// SIMATIC S7-200 project (STEP 7-Micro/WIN), CPU 222 REL 02.01

SYMBOL_TABLE USER1
CASSA_PIENA      C1       // CONTEGGIO DELLE DODICI BOTTIGLIE
FC_SUP           I0.0     // FINECORSA SUPERIORE
FC_INF           I0.1     // FINECORSA INFERIORE
FC_POS           I0.2     // SENSORE DI POSIZIONE
START            I0.3     // PULSANTE AVVIO CICLO
CONT             I0.4     // DISPOSITIVO CONTEGGIO BOTTIGLIE
IN_RIEMP         M0.0     // FASE DI RIEMPIMENTO
BOTT_OK          M0.2     // BOTTIGLIA DEPOSTA NELLA CASSA
DOSA             Q0.0     // DISPOSITIVO DI DOSAGGIO
IMP_INF          Q0.1     // DISPOSITIVO DI RIEMPIMENTO VERSO IL BASSO
IMP_SUP          Q0.2     // DISPOSITIVO DI RIEMPIMENTO VERSO L'ALTO
NASTRO           Q0.3     // NASTRO TRASPORTATORE
LAMP             Q0.4     // LAMPADA SPIA CONSENSO CICLO
T_FASE_RIEMP     T37      // TEMPO FSE DI RIEMPIMENTO
T_NUOVA          T39      // T PER L'INTRODUZIONE DI UNA NUOVA BOTTIGLIA
T_EVAQ           T40      // TEMPO EVAQUAZIONE DODICESIMA BOTTIGLIA
END_SYMBOL_TABLE

ORGANIZATION_BLOCK MAIN:OB1
TITLE=DPS 206 DISPOSITIVO DI IMBOTTIGLIAMENTO
BEGIN
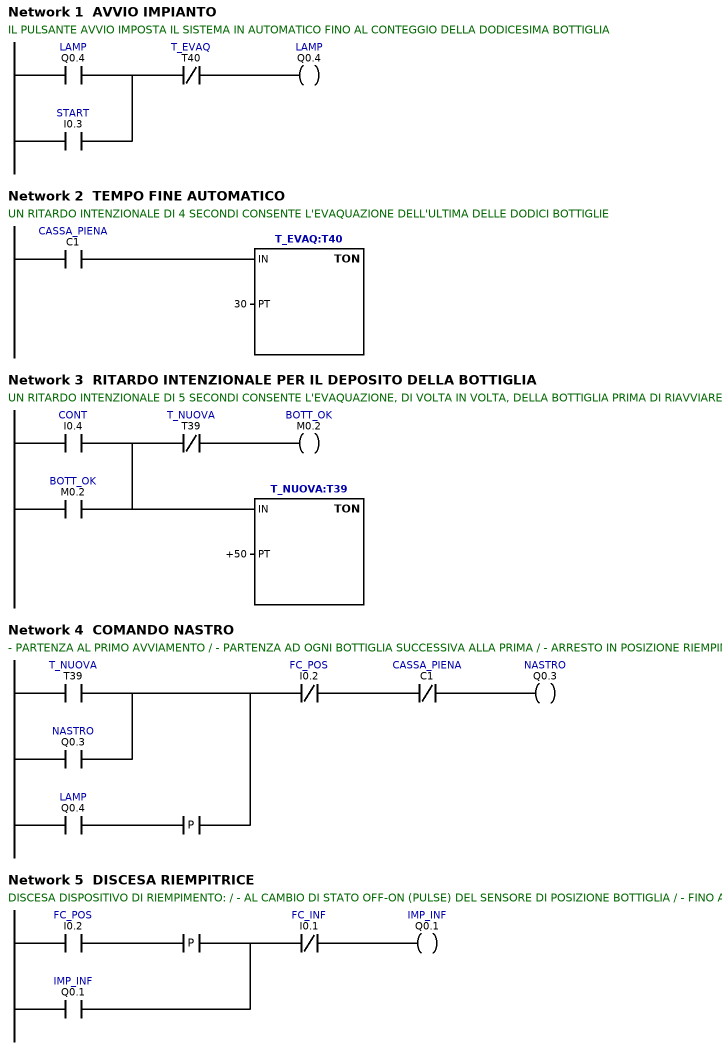
Network 1 // AVVIO IMPIANTO
// IL PULSANTE AVVIO IMPOSTA IL SISTEMA IN AUTOMATICO FINO AL CONTEGGIO DELLA DODICESIMA BOTTIGLIA
LD     LAMP:Q0.4
O      START:I0.3
AN     T_EVAQ:T40
=      LAMP:Q0.4
Network 2 // TEMPO FINE AUTOMATICO
// UN RITARDO INTENZIONALE DI 4 SECONDI CONSENTE L'EVAQUAZIONE DELL'ULTIMA DELLE DODICI BOTTIGLIE
LD     CASSA_PIENA:C1
TON    T_EVAQ:T40, 30
Network 3 // RITARDO INTENZIONALE PER IL DEPOSITO DELLA BOTTIGLIA
// UN RITARDO INTENZIONALE DI 5 SECONDI CONSENTE L'EVAQUAZIONE, DI VOLTA IN VOLTA, DELLA BOTTIGLIA PRIMA DI RIAVVIARE IL NASTRO
LD     CONT:I0.4
O      BOTT_OK:M0.2
LPS
AN     T_NUOVA:T39
=      BOTT_OK:M0.2
LPP
TON    T_NUOVA:T39, +50
Network 4 // COMANDO NASTRO
// - PARTENZA AL PRIMO AVVIAMENTO
// - PARTENZA AD OGNI BOTTIGLIA SUCCESSIVA ALLA PRIMA
// - ARRESTO IN POSIZIONE RIEMPIMENTO
// - ARRESTO A CASSA PIENA
LD     T_NUOVA:T39
O      NASTRO:Q0.3
LD     LAMP:Q0.4
EU
OLD
AN     FC_POS:I0.2
AN     CASSA_PIENA:C1
=      NASTRO:Q0.3
Network 5 // DISCESA RIEMPITRICE
// DISCESA DISPOSITIVO DI RIEMPIMENTO:
// - AL CAMBIO DI STATO OFF-ON (PULSE) DEL SENSORE DI POSIZIONE BOTTIGLIA
// - FINO AD IMPEGNARE IL FINECORSA INFERIORE FC_INF=ON
// 
LD     FC_POS:I0.2
EU
O      IMP_INF:Q0.1
AN     FC_INF:I0.1
=      IMP_INF:Q0.1
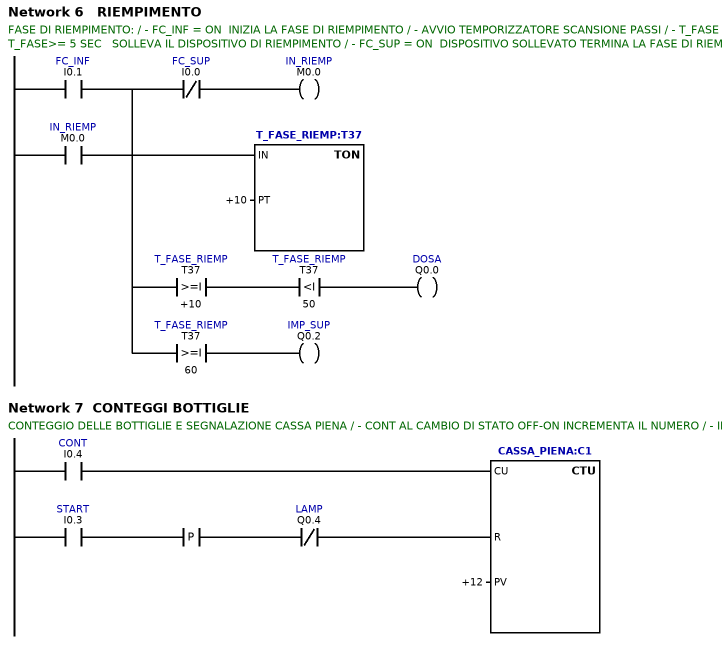
Network 6 //  RIEMPIMENTO
// FASE DI RIEMPIMENTO:
// - FC_INF = ON  INIZIA LA FASE DI RIEMPIMENTO
// - AVVIO TEMPORIZZATORE SCANSIONE PASSI
// - T_FASE >= 1 SEC  FINO A T_FASE < 4 SEC TIENE APERTO IL DOSATORE 
// - T_FASE>= 5 SEC   SOLLEVA IL DISPOSITIVO DI RIEMPIMENTO
// - FC_SUP = ON  DISPOSITIVO SOLLEVATO TERMINA LA FASE DI RIEMPIMENTO.
// 
LD     FC_INF:I0.1
O      IN_RIEMP:M0.0
LPS
AN     FC_SUP:I0.0
=      IN_RIEMP:M0.0
LRD
TON    T_FASE_RIEMP:T37, +10
LRD
AW>=   T_FASE_RIEMP:T37, +10
AW<    T_FASE_RIEMP:T37, 50
=      DOSA:Q0.0
LPP
AW>=   T_FASE_RIEMP:T37, 60
=      IMP_SUP:Q0.2
Network 7 // CONTEGGI BOTTIGLIE
// CONTEGGIO DELLE BOTTIGLIE E SEGNALAZIONE CASSA PIENA
// - CONT AL CAMBIO DI STATO OFF-ON INCREMENTA IL NUMERO
// - IL CONTEGGIO SI AZZERA AL RIAVVIO
LD     CONT:I0.4
LD     START:I0.3
EU
AN     LAMP:Q0.4
CTU    CASSA_PIENA:C1, +12
END_ORGANIZATION_BLOCK
